PROGRAM MAIN
VAR
	init : INT := 0;
END_VAR

HMILogic();
IF HMILogic.bRun = FALSE THEN
	Run.A_Man();
END_IF
IF HMILogic.bRun THEN
	Run(arrangedFrames := HMILogic.ArrangedFrames);
END_IF

END_PROGRAM

(* stored: Version 1.1.0.1, ProductVersion 3.1.4024.9
   POU MAIN: Id {6f26785d-3141-4d83-8f28-dd4e0f083bd8}, SpecialFunc None *)
